// Brief: Setup Arm Error Hold
FUNCTION_BLOCK PUBLIC FB_SetupCtrlDisable EXTENDS FB_SetupArmCtrlBase
VAR_INPUT
END_VAR
VAR_OUTPUT
END_VAR
VAR
END_VAR

END_FUNCTION_BLOCK

(* stored: Version 1.1.0.1, ProductVersion 3.1.4024.11
   POU FB_SetupCtrlDisable: Id {fd37dfd1-46dd-4a23-a295-d8873104bc66}, SpecialFunc None *)
